// TIA Portal V16 export
// export: Created 2023-06-21T17:06:27.3359127Z, ExportSetting WithDefaults, DisplayName Totally Integrated Automation Portal, DisplayVersion V16 Update 4, DisplayName TIA Portal Version Control Interface, DisplayVersion V16 Update 2, DisplayName TIA Portal Openness, DisplayVersion V16 Update 4, DisplayName SINAMICS Startdrive Advanced, DisplayVersion V16, DisplayName SINAMICS Startdrive G130, G150, S120, S150, SINAMICS MV, S210, DisplayVersion V16, DisplayName SINAMICS Startdrive G110M, G120, G120C, G120D, G120P, DisplayVersion V16, DisplayName STEP 7 Professional, DisplayVersion V16 Update 4, DisplayName STEP 7 Safety, DisplayVersion V16, DisplayName Soft Starter ES, DisplayVersion V16, DisplayName WinCC Advanced, DisplayVersion V16 Update 4
FUNCTION "Sts_Auto_Manual" : Void   // FC3, LAD
{ S7_Optimized_Access := 'TRUE' }
VERSION : 0.1
// stored: AutoNumber true, IsIECCheckEnabled false, SetENOAutomatically false, UDAEnableTagReadback false
   VAR_INPUT
      "30001" : Word;
   END_VAR
   VAR_TEMP
      Aux_1 : Word;
   END_VAR
BEGIN

REGION Network 1
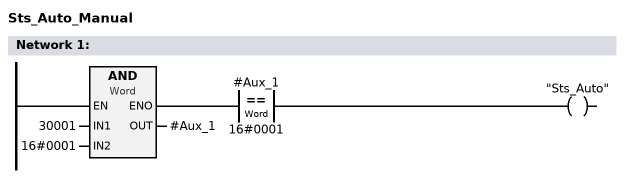
   RUNG wire#powerrail
      { S7_Templates := "SrcType := Word" } And(in1 := 30001, in2 := 16#0001, out => #Aux_1)
      { S7_Templates := "SrcType := Word" } EQ_Contact(in1 := #Aux_1, in2 := 16#0001)
      Coil( "Sts_Auto" )
   END_RUNG
   // the same network as SCL:
   #Aux_1 := 30001 AND 16#0001;
   "Sts_Auto" := #Aux_1 = 16#0001;
END_REGION
END_FUNCTION
